Staubli VAL3: session_get.pgx

program session_get(string& x_sName (dimensions=1))
  local num i
  local string l_sEmpty
  local string l_sEvent
begin
  //
  // get the actual session...
  //
  call saveData:getSession(x_sName)
  //
end
